PROGRAM MAIN
VAR
	input : ARRAY[0..4] OF LREAL := [1,1,1,1,1];	
	out : ARRAY[0..0] OF LREAL;
	FB_NN : FB_Dense_v1;

END_VAR

FB_NN(pointer_input := ADR(input),pointer_output:= ADR(out));

END_PROGRAM

(* stored: Version 1.1.0.1, ProductVersion 3.1.4024.12
   POU MAIN: Id {982bde0f-179e-4b17-b613-c9f5863bc8c6}, SpecialFunc None *)
